FUNCTION_BLOCK CAT1 (* Composite Function Block Type *)
  (* Standard: 61499-2 *)
  (* Version 0.0, 22/06/2021, Pranay Jhunjhunwala, Schneider Electric, template *)
  PACKAGE Main;
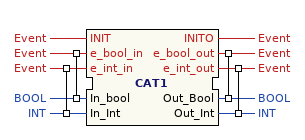
  EVENT_INPUT
    INIT; (* Initialization Request *)
    e_bool_in WITH In_bool; (* Normal Execution Request *)
    e_int_in WITH In_Int;
  END_EVENT
  EVENT_OUTPUT
    INITO; (* Initialization Confirm *)
    e_bool_out WITH Out_Bool; (* Execution Confirmation *)
    e_int_out WITH Out_Int;
  END_EVENT
  VAR_INPUT
    In_bool : BOOL; (* Input event qualifier *)
    In_Int : INT;
  END_VAR
  VAR_OUTPUT
    Out_Bool : BOOL; (* Output event qualifier *)
    Out_Int : INT;
  END_VAR
  FBS
    IThis : CAT1_HMI(QI := TRUE);
  END_FBS
  EVENT_CONNECTIONS
    INIT TO IThis.INIT;
    e_bool_in TO IThis.e_bool_in;
    e_int_in TO IThis.e_int_in;
    IThis.e_bool_out TO e_bool_out;
    IThis.e_int_out TO e_int_out;
    IThis.INITO TO INITO;
  END_CONNECTIONS
  DATA_CONNECTIONS
    In_bool TO IThis.hello;
    In_Int TO IThis.hello_int;
    IThis.out TO Out_Bool;
    IThis.out_int TO Out_Int;
  END_CONNECTIONS
END_FUNCTION_BLOCK
